FUNCTION_BLOCK E_D_FF
  (* Version 1.0, 2005-07-05, Goran Cengic, Chalmers *)
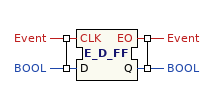
  EVENT_INPUT
    CLK WITH D;
  END_EVENT
  EVENT_OUTPUT
    EO WITH Q;
  END_EVENT
  VAR_INPUT
    D : BOOL;
  END_VAR
  VAR_OUTPUT
    Q : BOOL;
  END_VAR
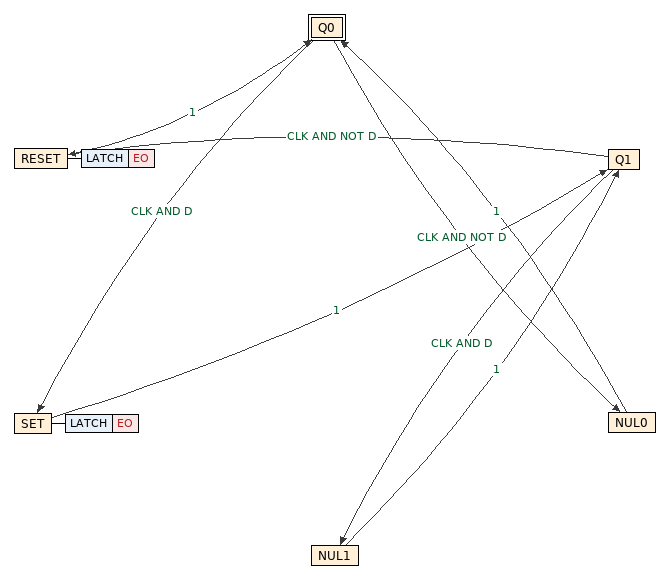
  EC_STATES
    Q0;
    Q1;
    NUL0;
    NUL1;
    SET : LATCH -> EO;
    RESET : LATCH -> EO;
  END_STATES
  EC_TRANSITIONS
    Q0 TO NUL0 := CLK AND NOT D;
    Q0 TO SET := CLK AND D;
    Q1 TO NUL1 := CLK AND D;
    Q1 TO RESET := CLK AND NOT D;
    SET TO Q1 := 1;
    RESET TO Q0 := 1;
    NUL0 TO Q0 := 1;
    NUL1 TO Q1 := 1;
  END_TRANSITIONS
  ALGORITHM LATCH IN Java:
Q = D;
  END_ALGORITHM
END_FUNCTION_BLOCK
